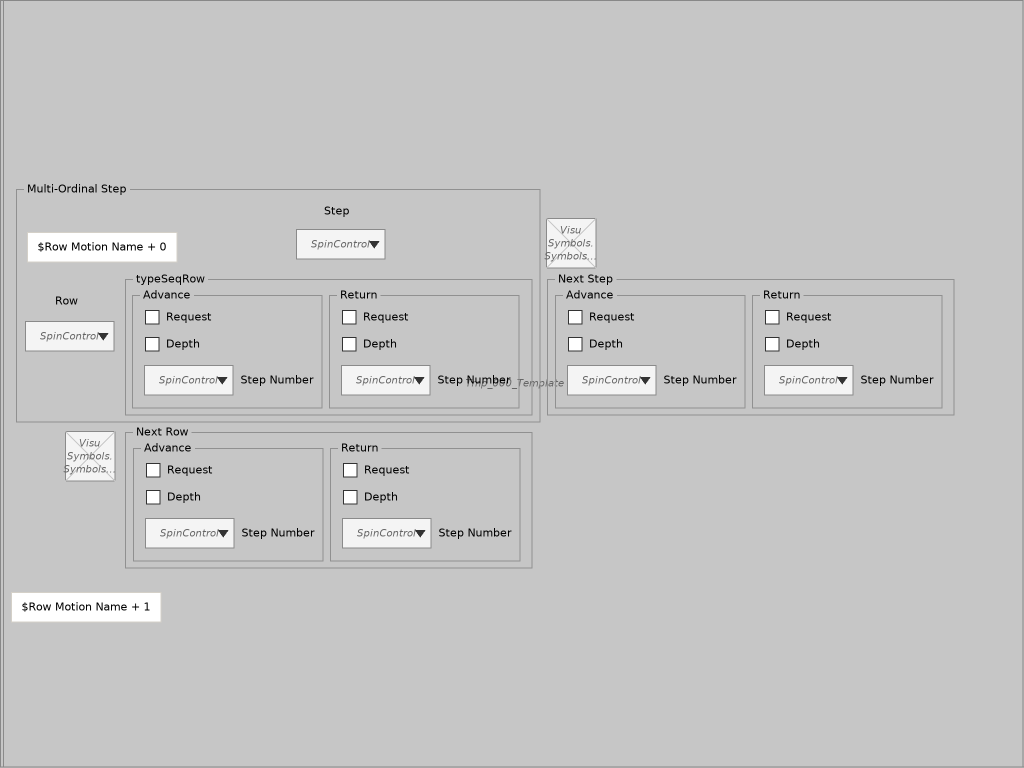
VISUALIZATION SeqTest  // 1024x768
    Frame (3,-1 1024x768)
        shows Tmp_000_Template(header := gHMIData.hmiHeader)
    GroupBox (16,181 524x241), "Multi-Ordinal Step"
        Textfield (11,51 150x30), "$Row Motion Name + 0"
    GroupBox (125,271 407x144), "typeSeqRow"
    GroupBox (329,287 190x121), "Return"
    GroupBox (132,287 190x121), "Advance"
    Label (202,365 150x30), "Step Number"
    Label (36,286 61x30), "Row"
    Label (295,196 84x30), "Step"
    SpinControl (25,321 89x30), variable: AutoRowsVisu.currentRowNum
        p651134158: AutoRows.numMaxMotionRows
        p1134531926: Row %d
    SpinControl (296,229 89x30), variable: AutoRowsVisu.currentStepNum
        p651134158: AutoRows.numMaxSeqSteps
        p1134531926: S %d
    Checkbox (143,302 150x30), "Request", variable: AutoRows.S1Seq.StationSequence[AutoRowsVisu.currentRowNum, AutoRowsVisu.currentStepNum].Advance.Request
    Checkbox (143,329 150x30), "Depth", variable: AutoRows.S1Seq.StationSequence[AutoRowsVisu.currentRowNum, AutoRowsVisu.currentStepNum].Advance.Depth
    SpinControl (144,365 89x30), variable: AutoRows.S1Seq.StationSequence[AutoRowsVisu.currentRowNum, AutoRowsVisu.currentStepNum].Advance.stepNumber
    Label (399,365 150x30), "Step Number"
    Checkbox (340,302 150x30), "Request", variable: AutoRows.S1Seq.StationSequence[AutoRowsVisu.currentRowNum, AutoRowsVisu.currentStepNum].Returnn.Request
    Checkbox (340,329 150x30), "Depth", variable: AutoRows.S1Seq.StationSequence[AutoRowsVisu.currentRowNum, AutoRowsVisu.currentStepNum].Returnn.Depth
    SpinControl (341,365 89x30), variable: AutoRows.S1Seq.StationSequence[AutoRowsVisu.currentRowNum, AutoRowsVisu.currentStepNum].Returnn.stepNumber
    GroupBox (125,424 407x144), "Next Row"
    GroupBox (330,440 190x121), "Return"
    GroupBox (133,440 190x121), "Advance"
    Label (203,518 150x30), "Step Number"
    Checkbox (144,455 150x30), "Request", variable: AutoRows.S1Seq.StationSequence[AutoRowsVisu.currentRowNum + 1, AutoRowsVisu.currentStepNum].Advance.Request
    Checkbox (144,482 150x30), "Depth", variable: AutoRows.S1Seq.StationSequence[AutoRowsVisu.currentRowNum + 1, AutoRowsVisu.currentStepNum].Advance.Depth
    SpinControl (145,518 89x30), variable: AutoRows.S1Seq.StationSequence[AutoRowsVisu.currentRowNum + 1, AutoRowsVisu.currentStepNum].Advance.stepNumber
    Label (400,518 150x30), "Step Number"
    Checkbox (341,455 150x30), "Request", variable: AutoRows.S1Seq.StationSequence[AutoRowsVisu.currentRowNum + 1, AutoRowsVisu.currentStepNum].Returnn.Request
    Checkbox (341,482 150x30), "Depth", variable: AutoRows.S1Seq.StationSequence[AutoRowsVisu.currentRowNum + 1, AutoRowsVisu.currentStepNum].Returnn.Depth
    SpinControl (342,518 89x30), variable: AutoRows.S1Seq.StationSequence[AutoRowsVisu.currentRowNum + 1, AutoRowsVisu.currentStepNum].Returnn.stepNumber
    Image (65,431 50x50), image: VisuSymbols.Symbols.ArrowBoldDown
    Image (546,218 50x50), image: VisuSymbols.Symbols.ArrowBoldRight
    GroupBox (547,271 407x144), "Next Step"
    GroupBox (752,287 190x121), "Return"
    GroupBox (555,287 190x121), "Advance"
    Label (625,365 150x30), "Step Number"
    Checkbox (566,302 150x30), "Request", variable: AutoRows.S1Seq.StationSequence[AutoRowsVisu.currentRowNum, AutoRowsVisu.currentStepNum + 1].Advance.Request
    Checkbox (566,329 150x30), "Depth", variable: AutoRows.S1Seq.StationSequence[AutoRowsVisu.currentRowNum, AutoRowsVisu.currentStepNum +1 ].Advance.Depth
    SpinControl (567,365 89x30), variable: AutoRows.S1Seq.StationSequence[AutoRowsVisu.currentRowNum, AutoRowsVisu.currentStepNum + 1].Advance.stepNumber
    Label (822,365 150x30), "Step Number"
    Checkbox (763,302 150x30), "Request", variable: AutoRows.S1Seq.StationSequence[AutoRowsVisu.currentRowNum, AutoRowsVisu.currentStepNum + 1].Returnn.Request
    Checkbox (763,329 150x30), "Depth", variable: AutoRows.S1Seq.StationSequence[AutoRowsVisu.currentRowNum, AutoRowsVisu.currentStepNum + 1].Returnn.Depth
    SpinControl (764,365 89x30), variable: AutoRows.S1Seq.StationSequence[AutoRowsVisu.currentRowNum, AutoRowsVisu.currentStepNum + 1].Returnn.stepNumber
    Textfield (11,592 150x30), "$Row Motion Name + 1"
END_VISUALIZATION

(* stored: Version 1.1.0.1, ProductVersion 3.1.4024.11
   Visu SeqTest: Id {a6d5374c-0559-086e-3847-d93dce919ea5} *)
